FUNCTION_BLOCK FB_ReadJsonReal
VAR_INPUT
	Member:STRING;
	sPath:STRING;
END_VAR
VAR_OUTPUT
	fReadValue:LREAL;
END_VAR
VAR
	nState: INT:=0;
	fbJsonDomParser:FB_JsonDomParser;
	ErrorCode :HRESULT;
	jSonProp :SJsonValue;
	jsonRoot :SJsonValue;
	bLoadDocument:BOOL;
END_VAR


CASE nState OF
	00: //Idle
		bLoadDocument:=FALSE;
		nState:=10;
		
	10: //Load the document
		bLoadDocument:=TRUE;
		fbJsonDomParser.LoadDocumentFromFile(sPath,bLoadDocument, hrErrorCode =>ErrorCode);
		IF ErrorCode = S_OK THEN
		nState:=20;
		END_IF
	
	20: //Read the desired values
		jsonRoot :=fbJsonDomParser.GetDocumentRoot();
		jSonProp := fbJsonDomParser.FindMember(jsonRoot,Member);
		IF (jsonProp<>0) THEN
			fReadValue := fbJsonDomParser.GetDouble(jSonProp);
		ELSE 
			fReadValue := -999999;
		END_IF
		
END_CASE

END_FUNCTION_BLOCK

(* stored: Version 1.1.0.1, ProductVersion 3.1.4024.14
   POU FB_ReadJsonReal: Id {4ba2a39c-a424-439c-a917-991d29f9a581}, SpecialFunc None *)
